FUNCTION_BLOCK ThreePhaseDevice
VAR_INPUT
	Ovld : BOOL;

END_VAR
VAR_OUTPUT
	Coil : BOOL;
END_VAR

VAR
	InternalFaultStatus : BOOL;
END_VAR

METHOD FaultRST : BOOL
VAR_INPUT
END_VAR
IF NOT Ovld THEN 
	FaultStatus := false;
END_IF
END_METHOD

METHOD FaultSet : BOOL
VAR_INPUT
END_VAR
IF Ovld THEN
	FaultStatus := TRUE;
END_IF
END_METHOD

PROPERTY FaultStatus : BOOL
GET
FaultStatus := InternalFaultStatus;
END_GET
SET
InternalFaultStatus := FaultStatus;
END_SET
END_PROPERTY

METHOD TurnOff : BOOL
VAR_INPUT
END_VAR
Coil := false;
END_METHOD

METHOD TurnOn : BOOL
VAR_INPUT
END_VAR
Coil := true;
END_METHOD

END_FUNCTION_BLOCK

(* stored: Version 1.1.0.1, ProductVersion 3.1.4024.15
   POU ThreePhaseDevice: Id {b8946281-48f9-4e67-9759-4dc34cb9618e}, SpecialFunc None
   Method FaultRST: Id {7c1e35fd-1691-43bf-a4cc-718fc81c26e2}
   Method FaultSet: Id {c185d64b-9c37-4ac4-b8a8-235e20ece85a}
   Property FaultStatus: Id {b593e086-5c8a-425e-9ea3-c68048df9c05}
   Get Get: Id {c8919eca-b2d3-43f1-9d09-1b51495fd21d}
   Set Set: Id {53ba1f5d-7f94-472a-8a8e-b3a56d0b88de}
   Method TurnOff: Id {da13e958-3919-44f8-952f-5d935d450d1b}
   Method TurnOn: Id {d33fd95f-05a3-4696-95ed-c288c7001f23} *)
